//A zone is occupied until the TU is handed over completly, or when the takeover is fully completed
FUNCTION F_PB_IsLogicalOccupied : BOOL
VAR_INPUT
	TransportControlData : REFERENCE TO ST_TransportControlData;
END_VAR
VAR
END_VAR


IF(NOT __ISVALIDREF(TransportControlData)) THEN RETURN; END_IF;

F_PB_IsLogicalOccupied := TransportControlData.Occupied OR TransportControlData.eTransportState = E_TransportState.HANDOVER;

END_FUNCTION

(* stored: Version 1.1.0.1, ProductVersion 3.1.4024.4
   POU F_PB_IsLogicalOccupied: Id {757800d9-2312-4648-93a0-64e370099057}, SpecialFunc None *)
